TYPE ST_SafetyZone :
STRUCT
	iNumber : INT;
	sName : STRING;
	bZoneTripped : BOOL; //Fed from TWINSAFE
END_STRUCT
END_TYPE

(* stored: Version 1.1.0.1, ProductVersion 3.1.4024.13
   DUT ST_SafetyZone: Id {a572f0c0-633e-4fc0-a2d3-92e64cc13c5c} *)
